// TwinCAT 3 PLC project PunchPLC1
// ProgramVersion: 3.1.4024.12
// libraries:
//   Tc2_Standard, * (Beckhoff Automation GmbH)
//   Tc2_System, * (Beckhoff Automation GmbH)
//   Tc3_Module, * (Beckhoff Automation GmbH)
// project tree:
//   GVLs/ GVL_HMI.TcGVL, GVL_IO.TcGVL, GVL_var.TcGVL
//   POUs/ FB_CasingVibratoryBowl1.TcPOU, FB_CoreVibratoryBowl2.TcPOU, MAIN.TcPOU, FB_OilPump.TcPOU, FB_CorePress.TcPOU, FB_CoreSwaging.TcPOU

// ---- GVLs/GVL_HMI.TcGVL
{attribute 'qualified_only'}
VAR_GLOBAL
	bCoreSwagingManualMode: BOOL := FALSE;
	sAlarmMessage: STRING(50) := '';
END_VAR

// ---- GVLs/GVL_IO.TcGVL
{attribute 'qualified_only'}
VAR_GLOBAL
	DI_24VDC_CB_OK 	AT %I*: BOOL := FALSE;
	DI_ESR1 		AT %I*: BOOL := FALSE;
	DI_M1 			AT %I*: BOOL := FALSE;
	DI_LS1	 		AT %I*: BOOL := FALSE;
	DI_TS1 			AT %I*: BOOL := FALSE;
	DI_CYL1_E 		AT %I*: BOOL := FALSE;
	DI_CYL1_R 		AT %I*: BOOL := FALSE;
	DI_CYL2_E 		AT %I*: BOOL := FALSE;
	DI_CYL2_R 		AT %I*: BOOL := FALSE;
	DI_CYL3_E 		AT %I*: BOOL := FALSE;
	DI_CYL3_R 		AT %I*: BOOL := FALSE;
	DI_CYL4_E 		AT %I*: BOOL := FALSE;
	DI_CYL4_R 		AT %I*: BOOL := FALSE;
	DI_CYL5_E 		AT %I*: BOOL := FALSE;
	DI_CYL5_R 		AT %I*: BOOL := FALSE;
	DI_CYL6_E 		AT %I*: BOOL := FALSE;
	DI_CYL6_R 		AT %I*: BOOL := FALSE;
	DI_CYL7_E 		AT %I*: BOOL := FALSE;
	DI_CYL7_R 		AT %I*: BOOL := FALSE;
	DI_PS1			AT %I*: BOOL := FALSE;
	DI_PCYL1_E		AT %I*: BOOL := FALSE;
	DI_PCYL1_R		AT %I*: BOOL := FALSE;
	DI_PCYL2_E		AT %I*: BOOL := FALSE;
	DI_PCYL2_R		AT %I*: BOOL := FALSE;
	DI_ECS			AT %I*: BOOL := FALSE;
	DI_EPD			AT %I*: BOOL := FALSE;
	DI_JLU			AT %I*: BOOL := FALSE;

	DI_PE1			AT %I*: BOOL := FALSE;
	DI_PE2			AT %I*: BOOL := FALSE;
	DI_PE3			AT %I*: BOOL := FALSE;
	DI_PE4			AT %I*: BOOL := FALSE;
	DI_PE5			AT %I*: BOOL := FALSE;
	DI_PE6			AT %I*: BOOL := FALSE;
	AI_PT1			AT %I*: REAL := 1.0;
	AI_PT2			AT %I*: REAL := 1.0;

	DO_M1			AT %Q*: BOOL;
	DO_M2			AT %Q*: BOOL;
	DO_VB1			AT %Q*: BOOL;
	DO_VB2			AT %Q*: BOOL;
	DO_SV1			AT %Q*: BOOL;
	DO_CYL1_E		AT %Q*: BOOL;
	DO_CYL1_R		AT %Q*: BOOL;
	DO_CYL2_E		AT %Q*: BOOL;
	DO_CYL2_R		AT %Q*: BOOL;
	DO_CYL3_E		AT %Q*: BOOL;
	DO_CYL3_R		AT %Q*: BOOL;
	DO_CYL4_E		AT %Q*: BOOL;
	DO_CYL4_R		AT %Q*: BOOL;
	DO_CYL5_E		AT %Q*: BOOL;
	DO_CYL5_R		AT %Q*: BOOL;
	DO_CYL6_E		AT %Q*: BOOL;
	DO_CYL6_R		AT %Q*: BOOL;
	DO_CYL7_E		AT %Q*: BOOL;
	DO_CYL7_R		AT %Q*: BOOL;
	DO_PCYL1_E		AT %Q*: BOOL;
	DO_PCYL1_R		AT %Q*: BOOL;
	DO_PCYL2_E		AT %Q*: BOOL;
	DO_PCYL2_R		AT %Q*: BOOL;
	DO_PCYL3_E		AT %Q*: BOOL;
	DO_PCYL4_E		AT %Q*: BOOL;
	DO_PCYL5_E		AT %Q*: BOOL;
	DO_PCYL6_E		AT %Q*: BOOL;
	DO_LGreen		AT %Q*: BOOL;
	DO_LRed			AT %Q*: BOOL;
END_VAR

// ---- GVLs/GVL_var.TcGVL
{attribute 'qualified_only'}
VAR_GLOBAL
	CorePress_CoreCount: INT := 0;
	CorePress_CasingCount: INT := 0;
	
	sAlarmMessage: STRING := "";
END_VAR

// ---- POUs/FB_CasingVibratoryBowl1.TcPOU
FUNCTION_BLOCK FB_CasingVibratoryBowl1
VAR_INPUT
    bEnable : BOOL;
    bReset : BOOL;
END_VAR

VAR_OUTPUT
	bFaulted: BOOL;
    iCasingCount : INT; (* Counts number of casings processed *)
END_VAR

VAR
    State : INT := 0;
    DelayTimer : TON;
END_VAR

CASE State OF
    0: (* Idle/Off *)
        IF GVL_IO.DI_24VDC_CB_OK AND GVL_IO.DI_ECS THEN
            State := 1;
        END_IF

    1: (* Wait for Product in Position *)
        DelayTimer(IN := TRUE, PT := T#50MS);
        IF DelayTimer.Q AND GVL_IO.DI_PE1 THEN
            State := 2;
        END_IF

    2: (* Energize Track Index Solenoid *)
        GVL_IO.DO_PCYL3_E := TRUE;
        DelayTimer(IN := TRUE, PT := T#250MS);
        IF DelayTimer.Q THEN
            GVL_IO.DO_PCYL3_E := FALSE;
            State := 3;
        END_IF

    3: (* Check Invert PE and Decide Path *)
        DelayTimer(IN := TRUE, PT := T#100MS);
        IF DelayTimer.Q THEN
            IF NOT GVL_IO.DI_PE2 THEN
                State := 5;
            ELSE
                State := 4;
            END_IF
        END_IF

    4: (* Energize Flipper Solenoid *)
        GVL_IO.DO_PCYL4_E := TRUE;
        DelayTimer(IN := TRUE, PT := T#150MS);
        IF DelayTimer.Q THEN
            GVL_IO.DO_PCYL4_E := FALSE;
            State := 6;
        END_IF

    5: (* Energize Straight Through Solenoid *)
        GVL_IO.DO_PCYL5_E := TRUE;
        DelayTimer(IN := TRUE, PT := T#250MS);
        IF DelayTimer.Q THEN
            GVL_IO.DO_PCYL5_E := FALSE;
            State := 2; (* Loop back *)
        END_IF

    6: (* Check High-Level Sensor *)
        DelayTimer(IN := TRUE, PT := T#500MS);
        IF DelayTimer.Q THEN
            IF GVL_IO.DI_PE4 THEN
                State := 6; (* Pause and wait *)
            ELSE
                iCasingCount := iCasingCount + 1;
                State := 2;
            END_IF
        END_IF
END_CASE

(* Reset logic *)
IF bReset THEN
    State := 0;
    iCasingCount := 0;
END_IF

END_FUNCTION_BLOCK

// ---- POUs/FB_CoreVibratoryBowl2.TcPOU
FUNCTION_BLOCK FB_CoreVibratoryBowl2
VAR_INPUT
    i_bEnabled : BOOL;
    i_bReset : BOOL;
END_VAR

VAR_OUTPUT
	o_bFaulted: BOOL;
    o_iCoreCount : INT; (* Counts number of cores processed *)
END_VAR

VAR
    iState : INT := 0;
    DelayTimer : TON;
END_VAR

CASE iState OF
    0: (* Idle/Off *)
        IF GVL_IO.DI_24VDC_CB_OK AND GVL_IO.DI_ECS THEN
            iState := 1;
        END_IF

    1: (* Wait for Product in Position *)
        DelayTimer(IN := TRUE, PT := T#50MS);
        IF DelayTimer.Q AND GVL_IO.DI_PE3 THEN
            iState := 2;
        END_IF

    2: (* Energize Core Track Index Solenoid *)
        GVL_IO.DO_PCYL6_E := TRUE;
        DelayTimer(IN := TRUE, PT := T#250MS);
        IF DelayTimer.Q THEN
            GVL_IO.DO_PCYL6_E := FALSE;
            iState := 3;
        END_IF

    3: (* Check High-Level Sensor *)
        DelayTimer(IN := TRUE, PT := T#500MS);
        IF DelayTimer.Q THEN
            IF GVL_IO.DI_PE6 THEN
                iState := 3; (* Pause and wait *)
            ELSE
                o_iCoreCount := o_iCoreCount + 1;
                iState := 2;
            END_IF
        END_IF
END_CASE

(* Reset logic *)
IF i_bReset THEN
    iState := 0;
    o_iCoreCount := 0;
END_IF

END_FUNCTION_BLOCK

// ---- POUs/MAIN.TcPOU
PROGRAM Main
VAR
	CoreSwaging: FB_CoreSwaging;
    OilPump: FB_OilPump;
    CorePress: FB_CorePress;
    CasingVibratoryBowl1: FB_CasingVibratoryBowl1;
    CoreVibratoryBowl2: FB_CoreVibratoryBowl2;

	bCoreSwagingFaulted: BOOL := FALSE;
	bOilPumpFaulted: BOOL := FALSE;
	bCorePressFaulted: BOOL := FALSE;
	bCasingVibratoryBowl1Faulted: BOOL := FALSE;
	bCoreVibratoryBowl2Faulted: BOOL := FALSE;
    bAnyRoutineFaulted: BOOL := FALSE;
END_VAR

IF NOT bAnyRoutineFaulted THEN
	CoreSwaging(i_bEnabled := TRUE);
	OilPump(i_bEnabled := TRUE);
	CorePress(i_bEnabled := TRUE);
	CasingVibratoryBowl1(i_bEnabled := TRUE);
	CoreVibratoryBowl2(i_bEnabled := TRUE);
	
	bCoreSwagingFaulted := CoreSwaging.o_bFaulted;
	bOilPumpFaulted := OilPump.o_bFaulted;
	bCorePressFaulted := CorePress.o_bFaulted;
	bCasingVibratoryBowl1Faulted := CasingVibratoryBowl1.o_bFaulted;
	bCoreVibratoryBowl2Faulted := CoreVibratoryBowl2.o_bFaulted;
	bAnyRoutineFaulted := bCoreSwagingFaulted OR bOilPumpFaulted
							OR bCorePressFaulted OR bCasingVibratoryBowl1Faulted OR bCoreVibratoryBowl2Faulted;
END_IF

GVL_IO.DO_LGreen := NOT bAnyRoutineFaulted;
GVL_IO.DO_LRed := bAnyRoutineFaulted;

END_PROGRAM

// ---- POUs/FB_CoreSwaging.TcPOU
FUNCTION_BLOCK FB_CoreSwaging
VAR_INPUT
	bEnable: BOOL;
    bReset : BOOL;  (* Reset from HMI *)
END_VAR
VAR_OUTPUT
	bFaulted: BOOL;
END_VAR
VAR
    State : INT := 0;
	FeedbackTimer : TON;
    DelayTimer : TON;
    AlarmTimer : TON;
    ManualMode : BOOL := FALSE;
    AlarmActive : BOOL := FALSE;
END_VAR

bFaulted := FALSE;

CASE State OF
	0: (* Idle/Off, DI_ECS=FALSE *)
		State := 10;
		
	10: (* check safety conditions *)
		IF GVL_IO.DI_24VDC_CB_OK AND GVL_IO.DI_ECS THEN (* Safeties OK and Enable Switch On *)
            GVL_IO.DO_M1 := TRUE; (* Start Oil Pump *)
			IF NOT DelayTimer.IN THEN
            	DelayTimer(IN := TRUE, PT := T#2S); (* 2 sec delay *)
			ELSE
				IF DelayTimer.Q AND GVL_IO.DI_M1 THEN
                	State := State + 10;
				END_IF
            END_IF
        END_IF
		
    20: (* Ensure CYL6 is Extended *)
        IF NOT GVL_IO.DI_CYL6_E THEN
            GVL_IO.DO_CYL6_E := TRUE;
        ELSE
            GVL_IO.DO_CYL6_E := FALSE;
            DelayTimer(IN := TRUE, PT := T#50MS);
            IF DelayTimer.Q THEN State := State + 1; END_IF
        END_IF
		
	21: (* Ensure CYL6 is Extended *)
    	IF NOT GVL_IO.DI_CYL5_R THEN
			GVL_IO.DO_CYL5_R := TRUE;
		ELSE
			GVL_IO.DO_CYL5_R := FALSE;
		END_IF
		
    30: (* Ensure CYL7 is Retracted *)
        IF NOT GVL_IO.DI_CYL7_R THEN
            GVL_IO.DO_CYL7_R := TRUE;
        ELSE
            GVL_IO.DO_CYL7_R := FALSE;
            DelayTimer(IN := TRUE, PT := T#50MS);
            IF DelayTimer.Q THEN State := State + 10; END_IF
        END_IF
    
    40: (* Low Lead Spool Check *)
        IF NOT GVL_IO.DI_PE5 THEN
            AlarmActive := TRUE;
            AlarmTimer(IN := TRUE, PT := T#3S);
        ELSE
            AlarmActive := FALSE;
            DelayTimer(IN := TRUE, PT := T#50MS);
            IF DelayTimer.Q THEN State := State + 10; END_IF
        END_IF
    
    50: (* Extend CYL7 *)
        IF NOT GVL_IO.DI_CYL7_E THEN
            GVL_IO.DO_CYL7_E := TRUE;
        ELSE
            GVL_IO.DO_CYL7_E := FALSE;
            DelayTimer(IN := TRUE, PT := T#50MS);
            IF DelayTimer.Q THEN State := State + 10; END_IF
        END_IF
    
    60: (* Retract CYL6 *)
        IF NOT GVL_IO.DI_CYL6_R THEN
            GVL_IO.DO_CYL6_R := TRUE;
        ELSE
            GVL_IO.DO_CYL6_R := FALSE;
            DelayTimer(IN := TRUE, PT := T#50MS);
            IF DelayTimer.Q THEN State := State + 10; END_IF
        END_IF
    
    70: (* Extend CYL5 *)
        IF NOT GVL_IO.DI_CYL5_E THEN
            GVL_IO.DO_CYL5_E := TRUE;
        ELSE
            GVL_IO.DO_CYL5_E := FALSE;
            DelayTimer(IN := TRUE, PT := T#250MS);
            IF DelayTimer.Q THEN State := State + 10; END_IF
        END_IF
    
    80: (* Retract CYL5 *)
        IF NOT GVL_IO.DI_CYL5_R THEN
            GVL_IO.DO_CYL5_R := TRUE;
        ELSE
            GVL_IO.DO_CYL5_R := FALSE;
            DelayTimer(IN := TRUE, PT := T#50MS);
            IF DelayTimer.Q THEN State := State + 10; END_IF
        END_IF
		
	90: (* Future Step *)
		State := 20;
END_CASE

(* Manual Mode Handling *)
IF ManualMode THEN
    State := 0; (* Hold state at 0 when in Manual Mode *)
    IF GVL_IO.DI_JLU THEN (* Jog switch pressed *)
        (* Motor M3 runs infinitely while switch is pressed *)
    END_IF
END_IF

(* Alarm Handling for Timeout *)
IF NOT AlarmActive AND (State > 0) THEN
    AlarmTimer(IN := FALSE);
ELSE
    IF AlarmTimer.Q THEN
        (* Trigger Alarm on HMI *)
    END_IF
END_IF

END_FUNCTION_BLOCK

// ---- POUs/FB_OilPump.TcPOU
FUNCTION_BLOCK FB_OilPump
VAR_INPUT
    bEnable : BOOL; (* Signal to enable the pump *)
    bReset : BOOL;  (* Reset signal from HMI *)
    bCallForCyl : BOOL; (* Any call for CYL1-CYL10 (DO5.6-DO6.3) *)
END_VAR

VAR_OUTPUT
    bFaulted : BOOL; (* Indicates failure to start alarm *)
END_VAR

VAR
    State : INT := 0; (* State machine variable *)
    StartDelayTimer : TON; (* Timer for 10s delay before activating DO5.2 *)
    FaultTimer : TON; (* Timer for 3s monitoring if DI1.3 feedback is missing *)
END_VAR

(* Default Output States *)
GVL_IO.DO_M1 := FALSE; (* Pump Primary Output *)
GVL_IO.DO_M2 := FALSE; (* Pump Secondary Output *)
GVL_IO.DO_SV1 := FALSE; (* Enable Pump if CYL is called *)
bFaulted := FALSE;

CASE State OF
    0: (* Pump Off, Not Enabled *)
        IF bEnable THEN
            State := 1;
        END_IF

    1: (* Pump Enabled from Other Routine *)
        GVL_IO.DO_M1 := TRUE; (* Start the pump *)
        
        (* Start the 10-second delay before DO5.2 activation *)
        StartDelayTimer(IN := TRUE, PT := T#10S);

        (* If delay timer completes, activate DO5.2 *)
        IF StartDelayTimer.Q THEN
            GVL_IO.DO_M2 := TRUE;
        END_IF

        (* Inhibit Pump if DI1.4 or DI1.5 goes Low *)
        IF (NOT GVL_IO.DI_LS1) OR (NOT GVL_IO.DI_TS1) THEN
            State := 2; (* Move to failure state *)
        END_IF

        (* If any CYL1-10 is called, Energise DO5.5 *)
        IF bCallForCyl THEN
            GVL_IO.DO_SV1 := TRUE;
        ELSE
            GVL_IO.DO_SV1 := FALSE;
        END_IF

    2: (* Fault Handling: Check DI1.3 Feedback *)
        (* Start 3-second timer to check for DI1.3 feedback *)
        FaultTimer(IN := TRUE, PT := T#3S);

        IF GVL_IO.DI_M1 THEN
            (* Reset fault condition if feedback is received in time *)
            FaultTimer(IN := FALSE);
            bFaulted := FALSE;
        END_IF

        IF FaultTimer.Q THEN
            (* If DI1.3 feedback was not received, set fault state *)
            bFaulted := TRUE;
        END_IF

        (* Reset Condition from HMI *)
        IF bReset THEN
            State := 0; (* Reset to the initial state *)
            FaultTimer(IN := FALSE);
            StartDelayTimer(IN := FALSE);
            bFaulted := FALSE;
        END_IF
END_CASE

END_FUNCTION_BLOCK

// ---- POUs/FB_CorePress.TcPOU
FUNCTION_BLOCK FB_CorePress
VAR_INPUT
    bEnable : BOOL; (* Enable the Core Press Sequence *)
    bReset : BOOL;  (* Reset from HMI *)
END_VAR

VAR_OUTPUT
    bFaulted : BOOL; (* Indicates failure alarm *)
    iProductCount : INT; (* Counts total cycles completed *)
END_VAR

VAR
    State : INT := 0;
    DelayTimer : TON;
    FaultTimer : TON;
END_VAR

CASE State OF
    0: (* Idle: Wait for safeties and enable switch *)
        IF GVL_IO.DI_24VDC_CB_OK AND GVL_IO.DI_ECS THEN
            State := 1;
        END_IF

    1: (* Start Oil Pump, Check Feedback *)
        GVL_IO.DO_M1 := TRUE; (* Start Oil Pump *)
        DelayTimer(IN := TRUE, PT := T#2S);
        
        IF DelayTimer.Q AND GVL_IO.DI_M1 THEN (* Feedback received *)
            State := 2;
        ELSE
            FaultTimer(IN := TRUE, PT := T#3S); (* Wait 3s for feedback *)
            IF FaultTimer.Q THEN
                bFaulted := TRUE; (* Alarm if no feedback *)
                State := 0;
            END_IF
        END_IF

    2: (* Check PCYL2 Retracted, Energize DO6.7 if needed *)
        IF NOT GVL_IO.DI_PCYL1_R THEN
            GVL_IO.DO_PCYL1_R := TRUE; (* Retract PCYL2 *)
        ELSE
            GVL_IO.DO_PCYL1_R := FALSE;
            State := 3;
        END_IF

    3: (* Count Casing/Core, Move to Next Step When Count Reached *)
        IF (GVL_Var.CorePress_CoreCount >= 5) AND (GVL_Var.CorePress_CasingCount >= 5) THEN
            State := 4;
        END_IF

    (* Continue adding logic for steps 4-11 as per your requirement *)

    11: (* Increment product count and loop back to step 2 *)
        iProductCount := iProductCount + 1;
        State := 2;
END_CASE

(* Reset logic *)
IF bReset THEN
    State := 0;
    bFaulted := FALSE;
    iProductCount := 0;
END_IF

END_FUNCTION_BLOCK
